// TIA Portal V17 export
// export: Created 2025-06-26T07:49:36.1041028Z, ExportSetting WithDefaults, DisplayName Totally Integrated Automation Portal, DisplayVersion V17 Update 8, DisplayName TIA Portal Openness, DisplayVersion V17 Update 8, DisplayName TIA Portal Version Control Interface, DisplayVersion V17, DisplayName STEP 7 Professional, DisplayVersion V17 Update 8, DisplayName STEP 7 Safety, DisplayVersion V17 Update 6, DisplayName WinCC Advanced, DisplayVersion V17 Update 8
FUNCTION_BLOCK "InputAlarmHandling"   // FB38, FBD
TITLE = Handle I/O alarms
{ S7_Optimized_Access := 'TRUE' }
AUTHOR : Heaten
VERSION : 0.1
// Handle I/O alarms
// stored: AutoNumber true, IsIECCheckEnabled false, IsRetainMemResEnabled false, MemoryReserve 0, SetENOAutomatically false, UDAEnableTagReadback false
   VAR
      A1102 { ExternalAccessible := 'False'; ExternalVisible := 'False'; ExternalWritable := 'False'; S7_SetPoint := 'True'} : "fbDigitalAlarm";
      A1103 { S7_SetPoint := 'True'} : "fbDigitalAlarm";
      A1110 { ExternalAccessible := 'False'; ExternalVisible := 'False'; ExternalWritable := 'False'; S7_SetPoint := 'True'} : "fbDigitalAlarm";
      A1122 { ExternalAccessible := 'False'; ExternalVisible := 'False'; ExternalWritable := 'False'; S7_SetPoint := 'True'} : "fbDigitalAlarm";
      A1123 { S7_SetPoint := 'True'} : "fbDigitalAlarm";
      A1130 { ExternalAccessible := 'False'; ExternalVisible := 'False'; ExternalWritable := 'False'; S7_SetPoint := 'True'} : "fbDigitalAlarm";
      A1142 { ExternalAccessible := 'False'; ExternalVisible := 'False'; ExternalWritable := 'False'; S7_SetPoint := 'True'} : "fbDigitalAlarm";
      A1143 { S7_SetPoint := 'True'} : "fbDigitalAlarm";
      A1150 { ExternalAccessible := 'False'; ExternalVisible := 'False'; ExternalWritable := 'False'; S7_SetPoint := 'True'} : "fbDigitalAlarm";
      A1201 { ExternalAccessible := 'False'; ExternalVisible := 'False'; ExternalWritable := 'False'; S7_SetPoint := 'True'} : "fbHMIEvent";
      A1202 { ExternalAccessible := 'False'; ExternalVisible := 'False'; ExternalWritable := 'False'; S7_SetPoint := 'True'} : "fbHMIEvent";
      A1203 { ExternalAccessible := 'False'; ExternalVisible := 'False'; ExternalWritable := 'False'; S7_SetPoint := 'True'} : "fbHMIEvent";
      A1204 { ExternalAccessible := 'False'; ExternalVisible := 'False'; ExternalWritable := 'False'; S7_SetPoint := 'True'} : "fbHMIEvent";
      A1205 { ExternalAccessible := 'False'; ExternalVisible := 'False'; ExternalWritable := 'False'; S7_SetPoint := 'True'} : "fbHMIEvent";
      A1206 { ExternalAccessible := 'False'; ExternalVisible := 'False'; ExternalWritable := 'False'; S7_SetPoint := 'True'} : "fbHMIEvent";
      A1207 { ExternalAccessible := 'False'; ExternalVisible := 'False'; ExternalWritable := 'False'; S7_SetPoint := 'True'} : "fbHMIEvent";
      A1208 { ExternalAccessible := 'False'; ExternalVisible := 'False'; ExternalWritable := 'False'; S7_SetPoint := 'True'} : "fbHMIEvent";
      A1209 { ExternalAccessible := 'False'; ExternalVisible := 'False'; ExternalWritable := 'False'; S7_SetPoint := 'True'} : "fbHMIEvent";
      A1210 { ExternalAccessible := 'False'; ExternalVisible := 'False'; ExternalWritable := 'False'; S7_SetPoint := 'True'} : "fbHMIEvent";
      A1212 { ExternalAccessible := 'False'; ExternalVisible := 'False'; ExternalWritable := 'False'; S7_SetPoint := 'True'} : "fbHMIEvent";
      A1213 { ExternalAccessible := 'False'; ExternalVisible := 'False'; ExternalWritable := 'False'; S7_SetPoint := 'True'} : "fbHMIEvent";
      A1214 { ExternalAccessible := 'False'; ExternalVisible := 'False'; ExternalWritable := 'False'; S7_SetPoint := 'True'} : "fbHMIEvent";
      A1215 { ExternalAccessible := 'False'; ExternalVisible := 'False'; ExternalWritable := 'False'; S7_SetPoint := 'True'} : "fbHMIEvent";
      A1220 { ExternalAccessible := 'False'; ExternalVisible := 'False'; ExternalWritable := 'False'; S7_SetPoint := 'True'} : "fbHMIEvent";
      A1221 { ExternalAccessible := 'False'; ExternalVisible := 'False'; ExternalWritable := 'False'; S7_SetPoint := 'True'} : "fbHMIEvent";
      A1223 { ExternalAccessible := 'False'; ExternalVisible := 'False'; ExternalWritable := 'False'; S7_SetPoint := 'True'} : "fbHMIEvent";
      A1231 { ExternalAccessible := 'False'; ExternalVisible := 'False'; ExternalWritable := 'False'; S7_SetPoint := 'True'} : "fbHMIEvent";
      A1232 { ExternalAccessible := 'False'; ExternalVisible := 'False'; ExternalWritable := 'False'; S7_SetPoint := 'True'} : "fbHMIEvent";
      A1233 { ExternalAccessible := 'False'; ExternalVisible := 'False'; ExternalWritable := 'False'; S7_SetPoint := 'True'} : "fbDigitalAlarm";
      A1241 { ExternalAccessible := 'False'; ExternalVisible := 'False'; ExternalWritable := 'False'; S7_SetPoint := 'True'} : "fbHMIEvent";
      A1242 { ExternalAccessible := 'False'; ExternalVisible := 'False'; ExternalWritable := 'False'; S7_SetPoint := 'True'} : "fbHMIEvent";
      A1243 { ExternalAccessible := 'False'; ExternalVisible := 'False'; ExternalWritable := 'False'; S7_SetPoint := 'True'} : "fbHMIEvent";
      A1244 { ExternalAccessible := 'False'; ExternalVisible := 'False'; ExternalWritable := 'False'; S7_SetPoint := 'True'} : "fbHMIEvent";
      A1255 { ExternalAccessible := 'False'; ExternalVisible := 'False'; ExternalWritable := 'False'; S7_SetPoint := 'True'} : "fbHMIEvent";
      A1256 { ExternalAccessible := 'False'; ExternalVisible := 'False'; ExternalWritable := 'False'; S7_SetPoint := 'True'} : "fbHMIEvent";
      A1257 { ExternalAccessible := 'False'; ExternalVisible := 'False'; ExternalWritable := 'False'; S7_SetPoint := 'True'} : "fbHMIEvent";
      A1264 { ExternalAccessible := 'False'; ExternalVisible := 'False'; ExternalWritable := 'False'; S7_SetPoint := 'True'} : "fbHMIEvent";
      A1266 { ExternalAccessible := 'False'; ExternalVisible := 'False'; ExternalWritable := 'False'; S7_SetPoint := 'True'} : "fbHMIEvent";
      A1267 { ExternalAccessible := 'False'; ExternalVisible := 'False'; ExternalWritable := 'False'; S7_SetPoint := 'True'} : "fbHMIEvent";
      A1268 { ExternalAccessible := 'False'; ExternalVisible := 'False'; ExternalWritable := 'False'; S7_SetPoint := 'True'} : "fbHMIEvent";
      A1274 { S7_SetPoint := 'True'} : "fbHMIEvent";
      A1276 { S7_SetPoint := 'True'} : "fbHMIEvent";
      A1277 { S7_SetPoint := 'True'} : "fbHMIEvent";
      A1278 { S7_SetPoint := 'True'} : "fbHMIEvent";
      A1279 { S7_SetPoint := 'True'} : "fbHMIEvent";
      A1280 { S7_SetPoint := 'True'} : "fbHMIEvent";
      A1281 { S7_SetPoint := 'True'} : "fbHMIEvent";
      A1282 { S7_SetPoint := 'True'} : "fbHMIEvent";
      A1283 { S7_SetPoint := 'True'} : "fbHMIEvent";
      A1284 { S7_SetPoint := 'True'} : "fbHMIEvent";
      A1285 { S7_SetPoint := 'True'} : "fbHMIEvent";
      A1286 { S7_SetPoint := 'True'} : "fbHMIEvent";
      A1287 { S7_SetPoint := 'True'} : "fbHMIEvent";
      A1288 { S7_SetPoint := 'True'} : "fbHMIEvent";
      A1289 { S7_SetPoint := 'True'} : "fbHMIEvent";
      A1290 { S7_SetPoint := 'True'} : "fbHMIEvent";
      A1291 { S7_SetPoint := 'True'} : "fbHMIEvent";
      A1292 { S7_SetPoint := 'True'} : "fbHMIEvent";
      A5250 { ExternalAccessible := 'False'; ExternalVisible := 'False'; ExternalWritable := 'False'; S7_SetPoint := 'True'} : "fbHMIEvent";
      A5251 { ExternalAccessible := 'False'; ExternalVisible := 'False'; ExternalWritable := 'False'; S7_SetPoint := 'True'} : "fbHMIEvent";
      A5252 { ExternalAccessible := 'False'; ExternalVisible := 'False'; ExternalWritable := 'False'; S7_SetPoint := 'True'} : "fbHMIEvent";
      A5253 { ExternalAccessible := 'False'; ExternalVisible := 'False'; ExternalWritable := 'False'; S7_SetPoint := 'True'} : "fbHMIEvent";
      A5254 { ExternalAccessible := 'False'; ExternalVisible := 'False'; ExternalWritable := 'False'; S7_SetPoint := 'True'} : "fbHMIEvent";
      A5255 { ExternalAccessible := 'False'; ExternalVisible := 'False'; ExternalWritable := 'False'; S7_SetPoint := 'True'} : "fbHMIEvent";
   END_VAR
BEGIN

REGION Network 1: 1102
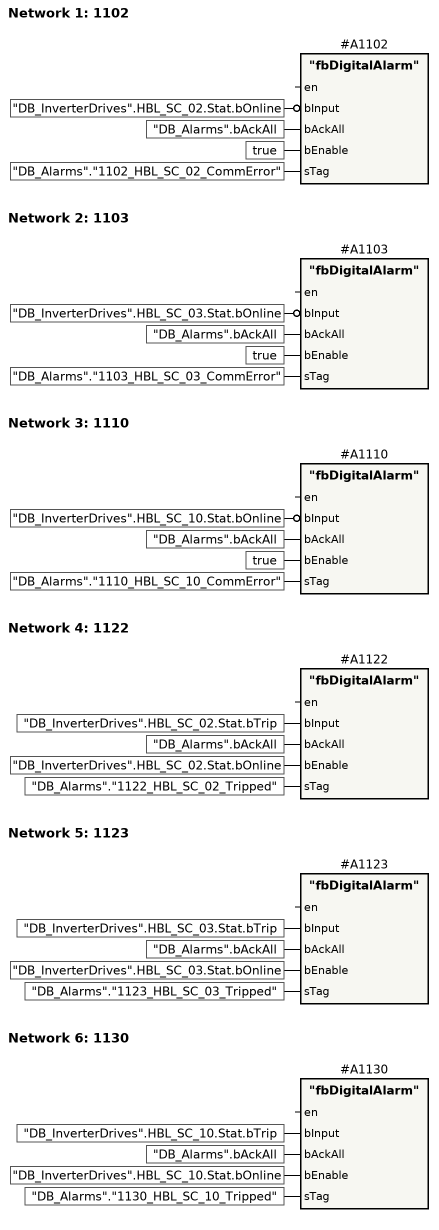
   #A1102(bInput := NOT "DB_InverterDrives".HBL_SC_02.Stat.bOnline,   // "fbDigitalAlarm"
          bAckAll := "DB_Alarms".bAckAll,
          bEnable := true,
          sTag := "DB_Alarms"."1102_HBL_SC_02_CommError");
END_REGION

REGION Network 2: 1103
   #A1103(bInput := NOT "DB_InverterDrives".HBL_SC_03.Stat.bOnline,   // "fbDigitalAlarm"
          bAckAll := "DB_Alarms".bAckAll,
          bEnable := true,
          sTag := "DB_Alarms"."1103_HBL_SC_03_CommError");
END_REGION

REGION Network 3: 1110
   #A1110(bInput := NOT "DB_InverterDrives".HBL_SC_10.Stat.bOnline,   // "fbDigitalAlarm"
          bAckAll := "DB_Alarms".bAckAll,
          bEnable := true,
          sTag := "DB_Alarms"."1110_HBL_SC_10_CommError");
END_REGION

REGION Network 4: 1122
   // Only show if online
   #A1122(bInput := "DB_InverterDrives".HBL_SC_02.Stat.bTrip,   // "fbDigitalAlarm"
          bAckAll := "DB_Alarms".bAckAll,
          bEnable := "DB_InverterDrives".HBL_SC_02.Stat.bOnline,
          sTag := "DB_Alarms"."1122_HBL_SC_02_Tripped");
END_REGION

REGION Network 5: 1123
   // Only show if online
   #A1123(bInput := "DB_InverterDrives".HBL_SC_03.Stat.bTrip,   // "fbDigitalAlarm"
          bAckAll := "DB_Alarms".bAckAll,
          bEnable := "DB_InverterDrives".HBL_SC_03.Stat.bOnline,
          sTag := "DB_Alarms"."1123_HBL_SC_03_Tripped");
END_REGION

REGION Network 6: 1130
   // Only show if online
   #A1130(bInput := "DB_InverterDrives".HBL_SC_10.Stat.bTrip,   // "fbDigitalAlarm"
          bAckAll := "DB_Alarms".bAckAll,
          bEnable := "DB_InverterDrives".HBL_SC_10.Stat.bOnline,
          sTag := "DB_Alarms"."1130_HBL_SC_10_Tripped");
END_REGION

REGION Network 7: 1142
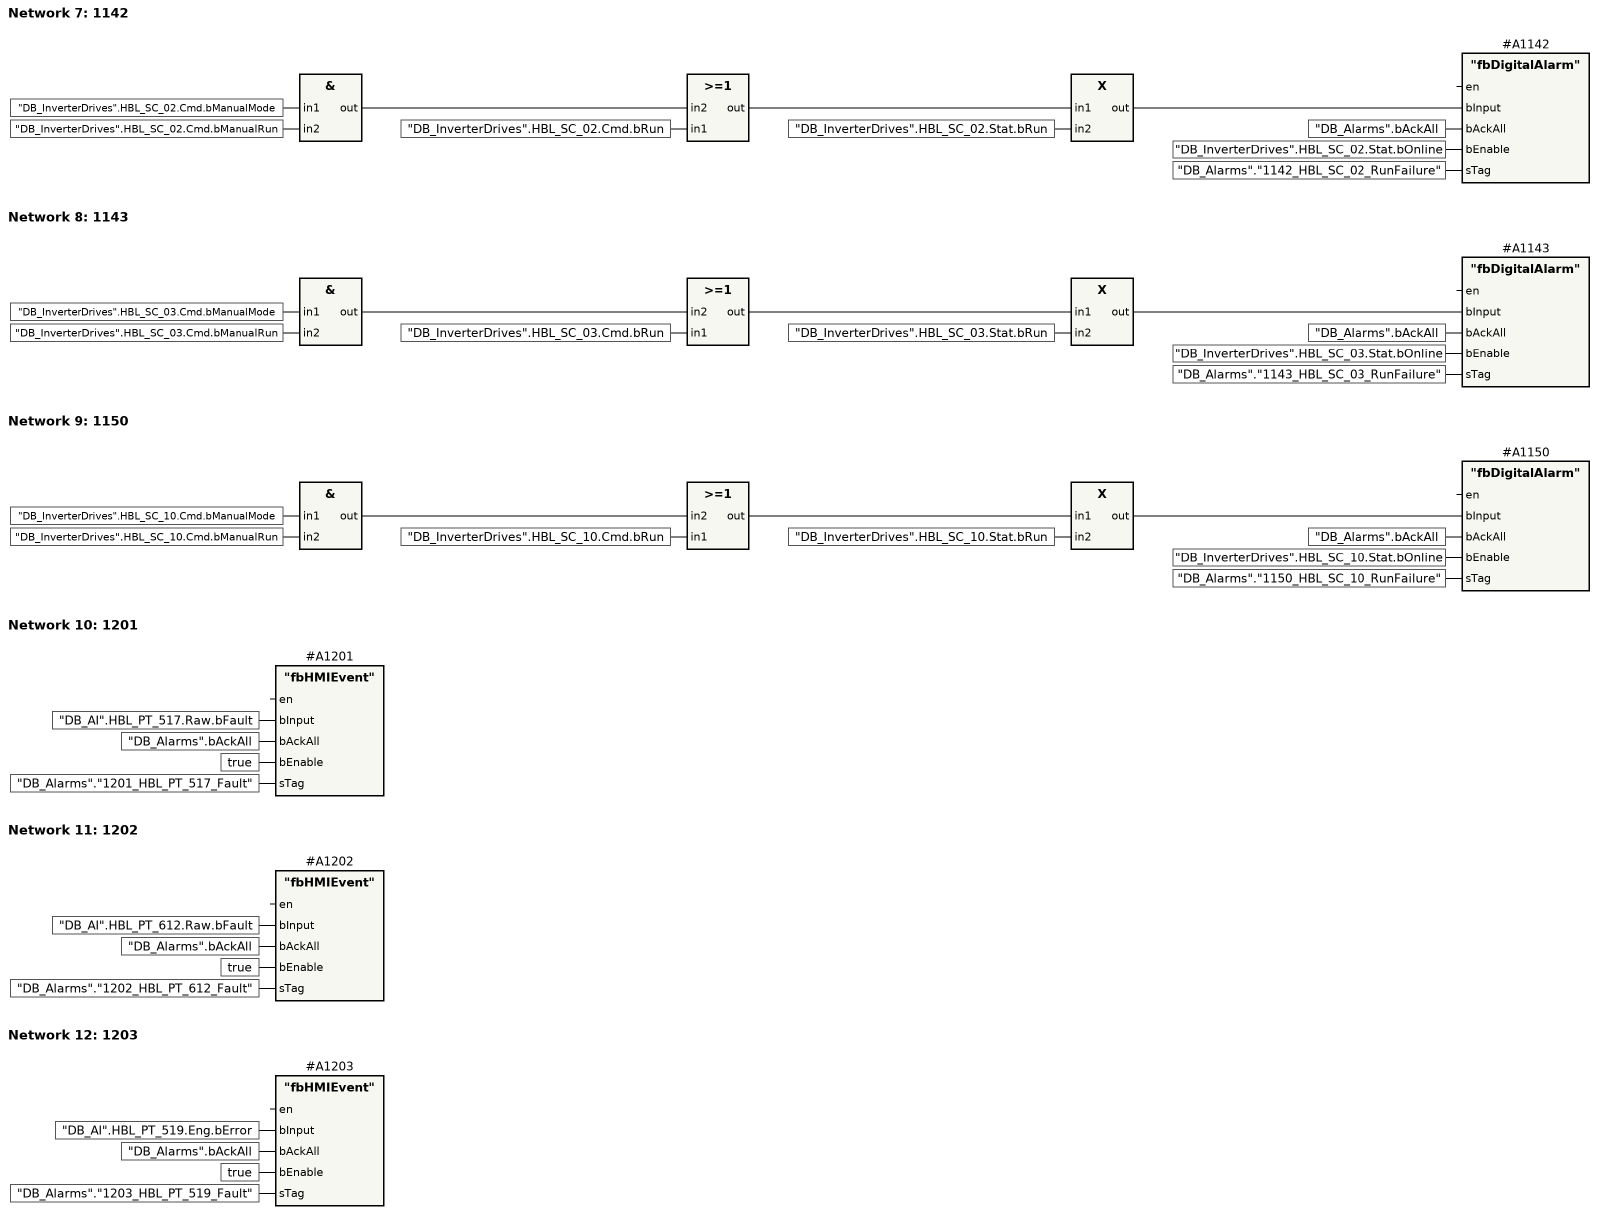
   #A1142(bInput := (("DB_InverterDrives".HBL_SC_02.Cmd.bManualMode AND "DB_InverterDrives".HBL_SC_02.Cmd.bManualRun) OR "DB_InverterDrives".HBL_SC_02.Cmd.bRun) XOR "DB_InverterDrives".HBL_SC_02.Stat.bRun,   // "fbDigitalAlarm"
          bAckAll := "DB_Alarms".bAckAll,
          bEnable := "DB_InverterDrives".HBL_SC_02.Stat.bOnline,
          sTag := "DB_Alarms"."1142_HBL_SC_02_RunFailure");
END_REGION

REGION Network 8: 1143
   #A1143(bInput := (("DB_InverterDrives".HBL_SC_03.Cmd.bManualMode AND "DB_InverterDrives".HBL_SC_03.Cmd.bManualRun) OR "DB_InverterDrives".HBL_SC_03.Cmd.bRun) XOR "DB_InverterDrives".HBL_SC_03.Stat.bRun,   // "fbDigitalAlarm"
          bAckAll := "DB_Alarms".bAckAll,
          bEnable := "DB_InverterDrives".HBL_SC_03.Stat.bOnline,
          sTag := "DB_Alarms"."1143_HBL_SC_03_RunFailure");
END_REGION

REGION Network 9: 1150
   #A1150(bInput := (("DB_InverterDrives".HBL_SC_10.Cmd.bManualMode AND "DB_InverterDrives".HBL_SC_10.Cmd.bManualRun) OR "DB_InverterDrives".HBL_SC_10.Cmd.bRun) XOR "DB_InverterDrives".HBL_SC_10.Stat.bRun,   // "fbDigitalAlarm"
          bAckAll := "DB_Alarms".bAckAll,
          bEnable := "DB_InverterDrives".HBL_SC_10.Stat.bOnline,
          sTag := "DB_Alarms"."1150_HBL_SC_10_RunFailure");
END_REGION

REGION Network 10: 1201
   #A1201(bInput := "DB_AI".HBL_PT_517.Raw.bFault,   // "fbHMIEvent"
          bAckAll := "DB_Alarms".bAckAll,
          bEnable := true,
          sTag := "DB_Alarms"."1201_HBL_PT_517_Fault");
END_REGION

REGION Network 11: 1202
   #A1202(bInput := "DB_AI".HBL_PT_612.Raw.bFault,   // "fbHMIEvent"
          bAckAll := "DB_Alarms".bAckAll,
          bEnable := true,
          sTag := "DB_Alarms"."1202_HBL_PT_612_Fault");
END_REGION

REGION Network 12: 1203
   #A1203(bInput := "DB_AI".HBL_PT_519.Eng.bError,   // "fbHMIEvent"
          bAckAll := "DB_Alarms".bAckAll,
          bEnable := true,
          sTag := "DB_Alarms"."1203_HBL_PT_519_Fault");
END_REGION

REGION Network 13: 1204
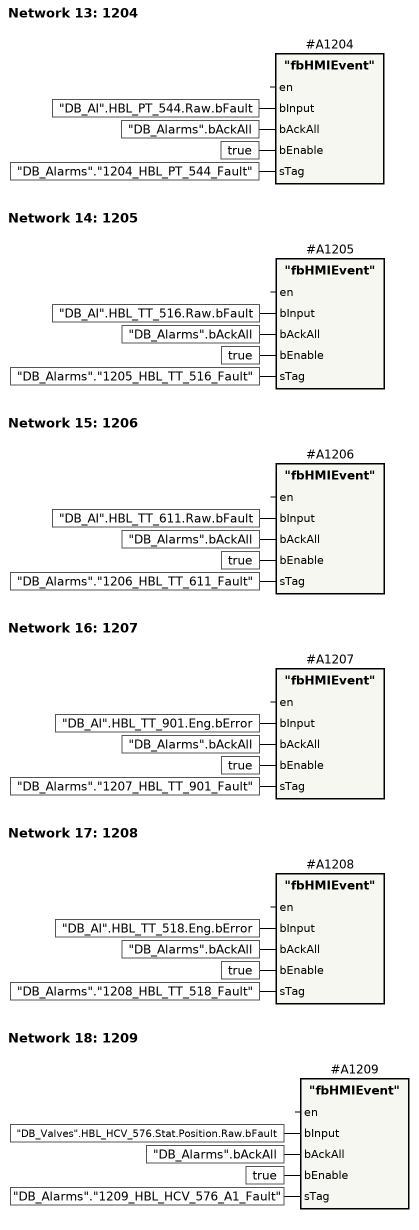
   #A1204(bInput := "DB_AI".HBL_PT_544.Raw.bFault,   // "fbHMIEvent"
          bAckAll := "DB_Alarms".bAckAll,
          bEnable := true,
          sTag := "DB_Alarms"."1204_HBL_PT_544_Fault");
END_REGION

REGION Network 14: 1205
   #A1205(bInput := "DB_AI".HBL_TT_516.Raw.bFault,   // "fbHMIEvent"
          bAckAll := "DB_Alarms".bAckAll,
          bEnable := true,
          sTag := "DB_Alarms"."1205_HBL_TT_516_Fault");
END_REGION

REGION Network 15: 1206
   #A1206(bInput := "DB_AI".HBL_TT_611.Raw.bFault,   // "fbHMIEvent"
          bAckAll := "DB_Alarms".bAckAll,
          bEnable := true,
          sTag := "DB_Alarms"."1206_HBL_TT_611_Fault");
END_REGION

REGION Network 16: 1207
   #A1207(bInput := "DB_AI".HBL_TT_901.Eng.bError,   // "fbHMIEvent"
          bAckAll := "DB_Alarms".bAckAll,
          bEnable := true,
          sTag := "DB_Alarms"."1207_HBL_TT_901_Fault");
END_REGION

REGION Network 17: 1208
   #A1208(bInput := "DB_AI".HBL_TT_518.Eng.bError,   // "fbHMIEvent"
          bAckAll := "DB_Alarms".bAckAll,
          bEnable := true,
          sTag := "DB_Alarms"."1208_HBL_TT_518_Fault");
END_REGION

REGION Network 18: 1209
   #A1209(bInput := "DB_Valves".HBL_HCV_576.Stat.Position.Raw.bFault,   // "fbHMIEvent"
          bAckAll := "DB_Alarms".bAckAll,
          bEnable := true,
          sTag := "DB_Alarms"."1209_HBL_HCV_576_A1_Fault");
END_REGION

REGION Network 19: 1210
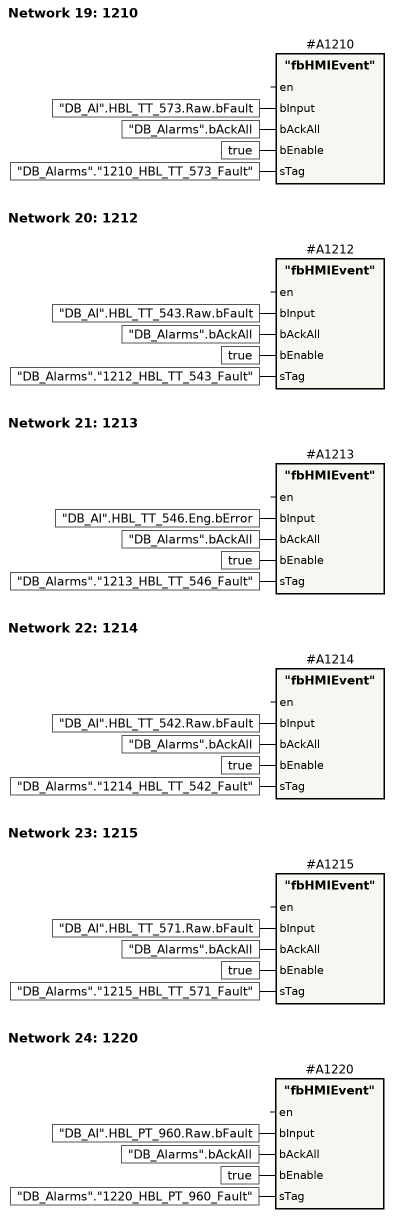
   #A1210(bInput := "DB_AI".HBL_TT_573.Raw.bFault,   // "fbHMIEvent"
          bAckAll := "DB_Alarms".bAckAll,
          bEnable := true,
          sTag := "DB_Alarms"."1210_HBL_TT_573_Fault");
END_REGION

REGION Network 20: 1212
   #A1212(bInput := "DB_AI".HBL_TT_543.Raw.bFault,   // "fbHMIEvent"
          bAckAll := "DB_Alarms".bAckAll,
          bEnable := true,
          sTag := "DB_Alarms"."1212_HBL_TT_543_Fault");
END_REGION

REGION Network 21: 1213
   #A1213(bInput := "DB_AI".HBL_TT_546.Eng.bError,   // "fbHMIEvent"
          bAckAll := "DB_Alarms".bAckAll,
          bEnable := true,
          sTag := "DB_Alarms"."1213_HBL_TT_546_Fault");
END_REGION

REGION Network 22: 1214
   #A1214(bInput := "DB_AI".HBL_TT_542.Raw.bFault,   // "fbHMIEvent"
          bAckAll := "DB_Alarms".bAckAll,
          bEnable := true,
          sTag := "DB_Alarms"."1214_HBL_TT_542_Fault");
END_REGION

REGION Network 23: 1215
   #A1215(bInput := "DB_AI".HBL_TT_571.Raw.bFault,   // "fbHMIEvent"
          bAckAll := "DB_Alarms".bAckAll,
          bEnable := true,
          sTag := "DB_Alarms"."1215_HBL_TT_571_Fault");
END_REGION

REGION Network 24: 1220
   #A1220(bInput := "DB_AI".HBL_PT_960.Raw.bFault,   // "fbHMIEvent"
          bAckAll := "DB_Alarms".bAckAll,
          bEnable := true,
          sTag := "DB_Alarms"."1220_HBL_PT_960_Fault");
END_REGION

REGION Network 25: 1221
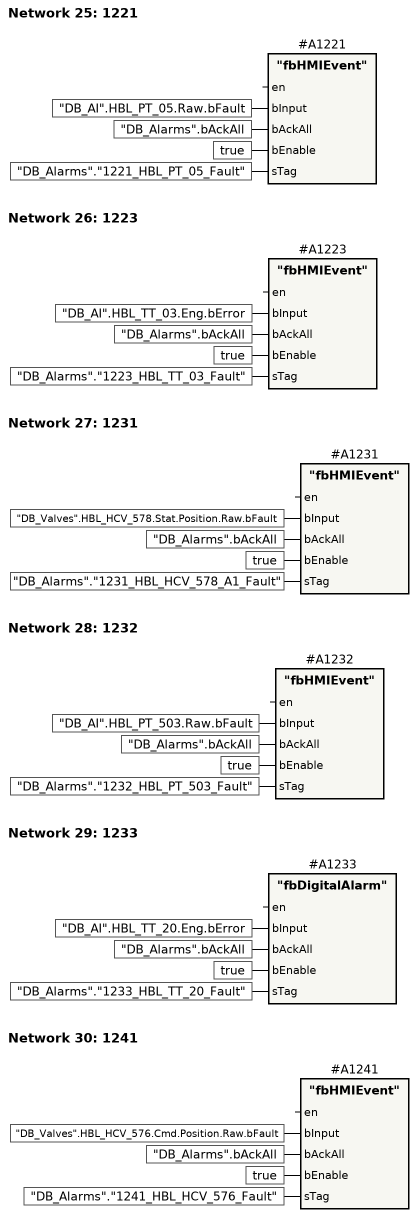
   #A1221(bInput := "DB_AI".HBL_PT_05.Raw.bFault,   // "fbHMIEvent"
          bAckAll := "DB_Alarms".bAckAll,
          bEnable := true,
          sTag := "DB_Alarms"."1221_HBL_PT_05_Fault");
END_REGION

REGION Network 26: 1223
   #A1223(bInput := "DB_AI".HBL_TT_03.Eng.bError,   // "fbHMIEvent"
          bAckAll := "DB_Alarms".bAckAll,
          bEnable := true,
          sTag := "DB_Alarms"."1223_HBL_TT_03_Fault");
END_REGION

REGION Network 27: 1231
   #A1231(bInput := "DB_Valves".HBL_HCV_578.Stat.Position.Raw.bFault,   // "fbHMIEvent"
          bAckAll := "DB_Alarms".bAckAll,
          bEnable := true,
          sTag := "DB_Alarms"."1231_HBL_HCV_578_A1_Fault");
END_REGION

REGION Network 28: 1232
   #A1232(bInput := "DB_AI".HBL_PT_503.Raw.bFault,   // "fbHMIEvent"
          bAckAll := "DB_Alarms".bAckAll,
          bEnable := true,
          sTag := "DB_Alarms"."1232_HBL_PT_503_Fault");
END_REGION

REGION Network 29: 1233
   #A1233(bInput := "DB_AI".HBL_TT_20.Eng.bError,   // "fbDigitalAlarm"
          bAckAll := "DB_Alarms".bAckAll,
          bEnable := true,
          sTag := "DB_Alarms"."1233_HBL_TT_20_Fault");
END_REGION

REGION Network 30: 1241
   #A1241(bInput := "DB_Valves".HBL_HCV_576.Cmd.Position.Raw.bFault,   // "fbHMIEvent"
          bAckAll := "DB_Alarms".bAckAll,
          bEnable := true,
          sTag := "DB_Alarms"."1241_HBL_HCV_576_Fault");
END_REGION

REGION Network 31: 1242
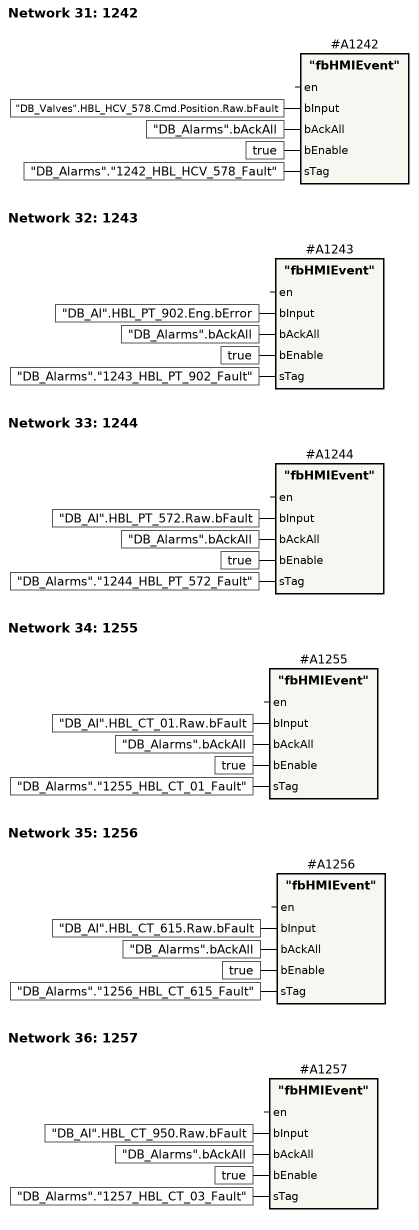
   #A1242(bInput := "DB_Valves".HBL_HCV_578.Cmd.Position.Raw.bFault,   // "fbHMIEvent"
          bAckAll := "DB_Alarms".bAckAll,
          bEnable := true,
          sTag := "DB_Alarms"."1242_HBL_HCV_578_Fault");
END_REGION

REGION Network 32: 1243
   #A1243(bInput := "DB_AI".HBL_PT_902.Eng.bError,   // "fbHMIEvent"
          bAckAll := "DB_Alarms".bAckAll,
          bEnable := true,
          sTag := "DB_Alarms"."1243_HBL_PT_902_Fault");
END_REGION

REGION Network 33: 1244
   #A1244(bInput := "DB_AI".HBL_PT_572.Raw.bFault,   // "fbHMIEvent"
          bAckAll := "DB_Alarms".bAckAll,
          bEnable := true,
          sTag := "DB_Alarms"."1244_HBL_PT_572_Fault");
END_REGION

REGION Network 34: 1255
   #A1255(bInput := "DB_AI".HBL_CT_01.Raw.bFault,   // "fbHMIEvent"
          bAckAll := "DB_Alarms".bAckAll,
          bEnable := true,
          sTag := "DB_Alarms"."1255_HBL_CT_01_Fault");
END_REGION

REGION Network 35: 1256
   #A1256(bInput := "DB_AI".HBL_CT_615.Raw.bFault,   // "fbHMIEvent"
          bAckAll := "DB_Alarms".bAckAll,
          bEnable := true,
          sTag := "DB_Alarms"."1256_HBL_CT_615_Fault");
END_REGION

REGION Network 36: 1257
   #A1257(bInput := "DB_AI".HBL_CT_950.Raw.bFault,   // "fbHMIEvent"
          bAckAll := "DB_Alarms".bAckAll,
          bEnable := true,
          sTag := "DB_Alarms"."1257_HBL_CT_03_Fault");
END_REGION

REGION Network 37: 1264
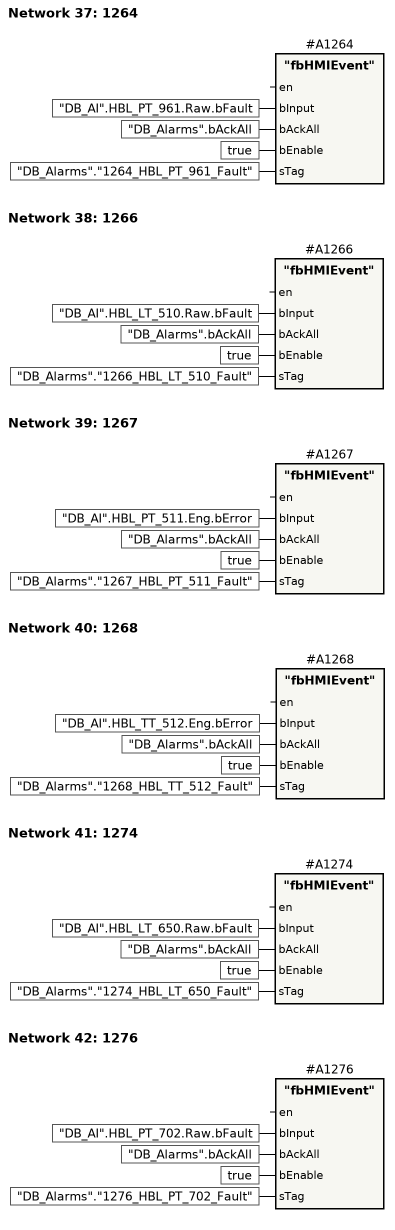
   #A1264(bInput := "DB_AI".HBL_PT_961.Raw.bFault,   // "fbHMIEvent"
          bAckAll := "DB_Alarms".bAckAll,
          bEnable := true,
          sTag := "DB_Alarms"."1264_HBL_PT_961_Fault");
END_REGION

REGION Network 38: 1266
   #A1266(bInput := "DB_AI".HBL_LT_510.Raw.bFault,   // "fbHMIEvent"
          bAckAll := "DB_Alarms".bAckAll,
          bEnable := true,
          sTag := "DB_Alarms"."1266_HBL_LT_510_Fault");
END_REGION

REGION Network 39: 1267
   #A1267(bInput := "DB_AI".HBL_PT_511.Eng.bError,   // "fbHMIEvent"
          bAckAll := "DB_Alarms".bAckAll,
          bEnable := true,
          sTag := "DB_Alarms"."1267_HBL_PT_511_Fault");
END_REGION

REGION Network 40: 1268
   #A1268(bInput := "DB_AI".HBL_TT_512.Eng.bError,   // "fbHMIEvent"
          bAckAll := "DB_Alarms".bAckAll,
          bEnable := true,
          sTag := "DB_Alarms"."1268_HBL_TT_512_Fault");
END_REGION

REGION Network 41: 1274
   #A1274(bInput := "DB_AI".HBL_LT_650.Raw.bFault,   // "fbHMIEvent"
          bAckAll := "DB_Alarms".bAckAll,
          bEnable := true,
          sTag := "DB_Alarms"."1274_HBL_LT_650_Fault");
END_REGION

REGION Network 42: 1276
   #A1276(bInput := "DB_AI".HBL_PT_702.Raw.bFault,   // "fbHMIEvent"
          bAckAll := "DB_Alarms".bAckAll,
          bEnable := true,
          sTag := "DB_Alarms"."1276_HBL_PT_702_Fault");
END_REGION

REGION Network 43: 1277
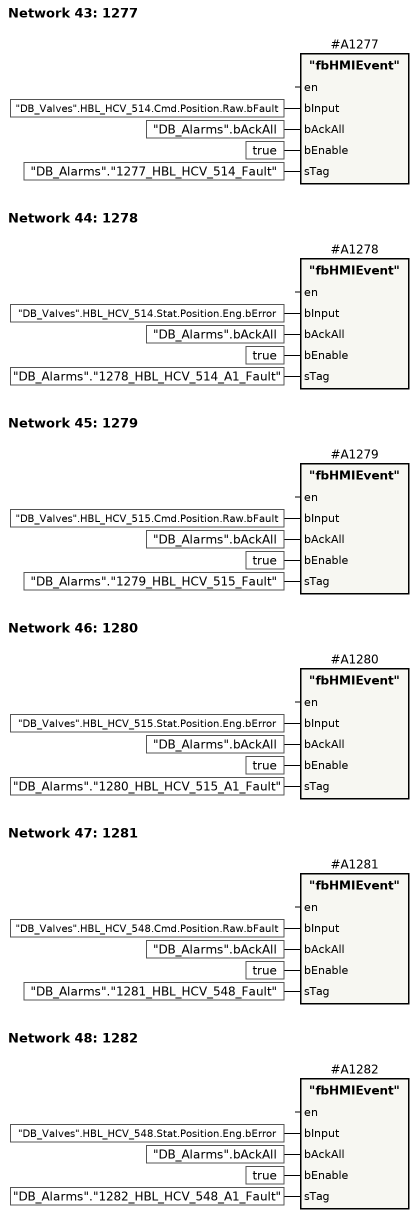
   #A1277(bInput := "DB_Valves".HBL_HCV_514.Cmd.Position.Raw.bFault,   // "fbHMIEvent"
          bAckAll := "DB_Alarms".bAckAll,
          bEnable := true,
          sTag := "DB_Alarms"."1277_HBL_HCV_514_Fault");
END_REGION

REGION Network 44: 1278
   #A1278(bInput := "DB_Valves".HBL_HCV_514.Stat.Position.Eng.bError,   // "fbHMIEvent"
          bAckAll := "DB_Alarms".bAckAll,
          bEnable := true,
          sTag := "DB_Alarms"."1278_HBL_HCV_514_A1_Fault");
END_REGION

REGION Network 45: 1279
   #A1279(bInput := "DB_Valves".HBL_HCV_515.Cmd.Position.Raw.bFault,   // "fbHMIEvent"
          bAckAll := "DB_Alarms".bAckAll,
          bEnable := true,
          sTag := "DB_Alarms"."1279_HBL_HCV_515_Fault");
END_REGION

REGION Network 46: 1280
   #A1280(bInput := "DB_Valves".HBL_HCV_515.Stat.Position.Eng.bError,   // "fbHMIEvent"
          bAckAll := "DB_Alarms".bAckAll,
          bEnable := true,
          sTag := "DB_Alarms"."1280_HBL_HCV_515_A1_Fault");
END_REGION

REGION Network 47: 1281
   #A1281(bInput := "DB_Valves".HBL_HCV_548.Cmd.Position.Raw.bFault,   // "fbHMIEvent"
          bAckAll := "DB_Alarms".bAckAll,
          bEnable := true,
          sTag := "DB_Alarms"."1281_HBL_HCV_548_Fault");
END_REGION

REGION Network 48: 1282
   #A1282(bInput := "DB_Valves".HBL_HCV_548.Stat.Position.Eng.bError,   // "fbHMIEvent"
          bAckAll := "DB_Alarms".bAckAll,
          bEnable := true,
          sTag := "DB_Alarms"."1282_HBL_HCV_548_A1_Fault");
END_REGION

REGION Network 49: 1283
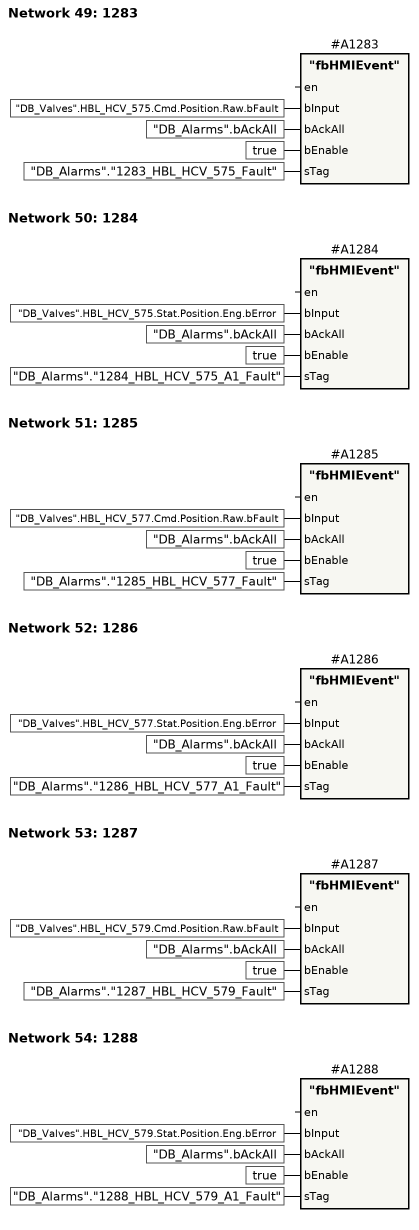
   #A1283(bInput := "DB_Valves".HBL_HCV_575.Cmd.Position.Raw.bFault,   // "fbHMIEvent"
          bAckAll := "DB_Alarms".bAckAll,
          bEnable := true,
          sTag := "DB_Alarms"."1283_HBL_HCV_575_Fault");
END_REGION

REGION Network 50: 1284
   #A1284(bInput := "DB_Valves".HBL_HCV_575.Stat.Position.Eng.bError,   // "fbHMIEvent"
          bAckAll := "DB_Alarms".bAckAll,
          bEnable := true,
          sTag := "DB_Alarms"."1284_HBL_HCV_575_A1_Fault");
END_REGION

REGION Network 51: 1285
   #A1285(bInput := "DB_Valves".HBL_HCV_577.Cmd.Position.Raw.bFault,   // "fbHMIEvent"
          bAckAll := "DB_Alarms".bAckAll,
          bEnable := true,
          sTag := "DB_Alarms"."1285_HBL_HCV_577_Fault");
END_REGION

REGION Network 52: 1286
   #A1286(bInput := "DB_Valves".HBL_HCV_577.Stat.Position.Eng.bError,   // "fbHMIEvent"
          bAckAll := "DB_Alarms".bAckAll,
          bEnable := true,
          sTag := "DB_Alarms"."1286_HBL_HCV_577_A1_Fault");
END_REGION

REGION Network 53: 1287
   #A1287(bInput := "DB_Valves".HBL_HCV_579.Cmd.Position.Raw.bFault,   // "fbHMIEvent"
          bAckAll := "DB_Alarms".bAckAll,
          bEnable := true,
          sTag := "DB_Alarms"."1287_HBL_HCV_579_Fault");
END_REGION

REGION Network 54: 1288
   #A1288(bInput := "DB_Valves".HBL_HCV_579.Stat.Position.Eng.bError,   // "fbHMIEvent"
          bAckAll := "DB_Alarms".bAckAll,
          bEnable := true,
          sTag := "DB_Alarms"."1288_HBL_HCV_579_A1_Fault");
END_REGION

REGION Network 55: 1289
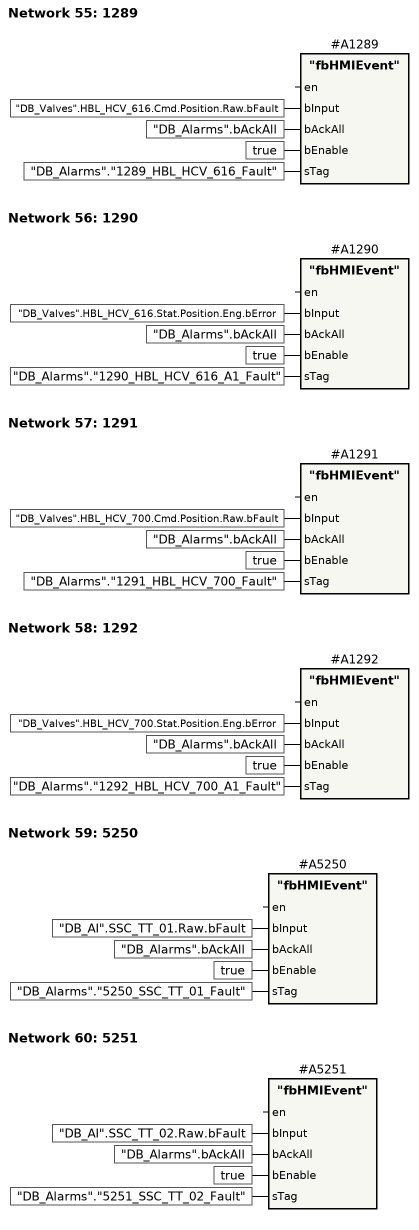
   #A1289(bInput := "DB_Valves".HBL_HCV_616.Cmd.Position.Raw.bFault,   // "fbHMIEvent"
          bAckAll := "DB_Alarms".bAckAll,
          bEnable := true,
          sTag := "DB_Alarms"."1289_HBL_HCV_616_Fault");
END_REGION

REGION Network 56: 1290
   #A1290(bInput := "DB_Valves".HBL_HCV_616.Stat.Position.Eng.bError,   // "fbHMIEvent"
          bAckAll := "DB_Alarms".bAckAll,
          bEnable := true,
          sTag := "DB_Alarms"."1290_HBL_HCV_616_A1_Fault");
END_REGION

REGION Network 57: 1291
   #A1291(bInput := "DB_Valves".HBL_HCV_700.Cmd.Position.Raw.bFault,   // "fbHMIEvent"
          bAckAll := "DB_Alarms".bAckAll,
          bEnable := true,
          sTag := "DB_Alarms"."1291_HBL_HCV_700_Fault");
END_REGION

REGION Network 58: 1292
   #A1292(bInput := "DB_Valves".HBL_HCV_700.Stat.Position.Eng.bError,   // "fbHMIEvent"
          bAckAll := "DB_Alarms".bAckAll,
          bEnable := true,
          sTag := "DB_Alarms"."1292_HBL_HCV_700_A1_Fault");
END_REGION

REGION Network 59: 5250
   #A5250(bInput := "DB_AI".SSC_TT_01.Raw.bFault,   // "fbHMIEvent"
          bAckAll := "DB_Alarms".bAckAll,
          bEnable := true,
          sTag := "DB_Alarms"."5250_SSC_TT_01_Fault");
END_REGION

REGION Network 60: 5251
   #A5251(bInput := "DB_AI".SSC_TT_02.Raw.bFault,   // "fbHMIEvent"
          bAckAll := "DB_Alarms".bAckAll,
          bEnable := true,
          sTag := "DB_Alarms"."5251_SSC_TT_02_Fault");
END_REGION

REGION Network 61: 5252
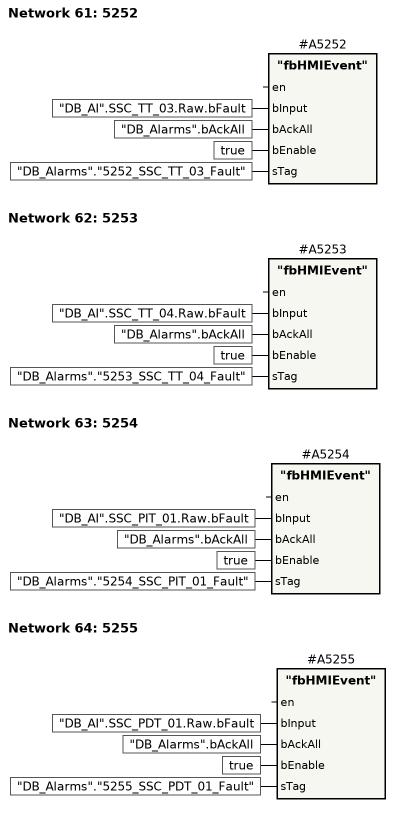
   #A5252(bInput := "DB_AI".SSC_TT_03.Raw.bFault,   // "fbHMIEvent"
          bAckAll := "DB_Alarms".bAckAll,
          bEnable := true,
          sTag := "DB_Alarms"."5252_SSC_TT_03_Fault");
END_REGION

REGION Network 62: 5253
   #A5253(bInput := "DB_AI".SSC_TT_04.Raw.bFault,   // "fbHMIEvent"
          bAckAll := "DB_Alarms".bAckAll,
          bEnable := true,
          sTag := "DB_Alarms"."5253_SSC_TT_04_Fault");
END_REGION

REGION Network 63: 5254
   #A5254(bInput := "DB_AI".SSC_PIT_01.Raw.bFault,   // "fbHMIEvent"
          bAckAll := "DB_Alarms".bAckAll,
          bEnable := true,
          sTag := "DB_Alarms"."5254_SSC_PIT_01_Fault");
END_REGION

REGION Network 64: 5255
   #A5255(bInput := "DB_AI".SSC_PDT_01.Raw.bFault,   // "fbHMIEvent"
          bAckAll := "DB_Alarms".bAckAll,
          bEnable := true,
          sTag := "DB_Alarms"."5255_SSC_PDT_01_Fault");
END_REGION
END_FUNCTION_BLOCK
